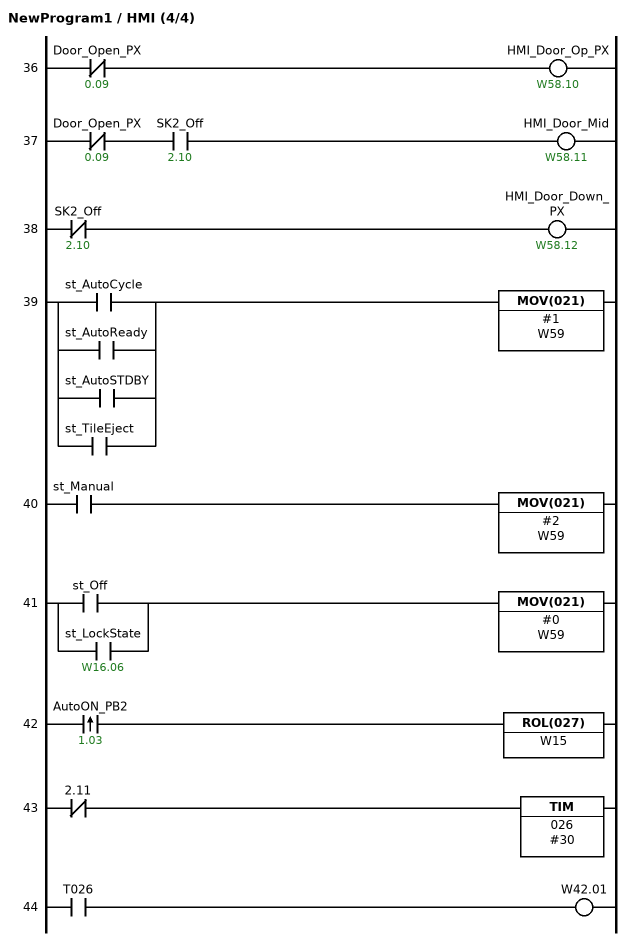
; [picture p48: NewProgram1 / HMI, rungs 36-44]
; rung 36
LDNOT Door_Open_PX  ; 0.09
OUT HMI_Door_Op_PX  ; W58.10
; rung 37
LDNOT Door_Open_PX  ; 0.09
AND SK2_Off  ; 2.10
OUT HMI_Door_Mid  ; W58.11
; rung 38
LDNOT SK2_Off  ; 2.10
OUT HMI_Door_Down_PX  ; W58.12
; rung 39
LD st_AutoCycle
OR st_AutoReady
OR st_AutoSTDBY
OR st_TileEject
MOV(021) #1 W59
; rung 40
LD st_Manual
MOV(021) #2 W59
; rung 41
LD st_Off
OR st_LockState  ; W16.06
MOV(021) #0 W59
; rung 42
@LD AutoON_PB2  ; 1.03
ROL(027) W15
; rung 43
LDNOT 2.11
TIM 026 #30
; rung 44
LD T026
OUT W42.01

### Section END
; rung 0
END(001)